// TIA Portal V18 export
FUNCTION_BLOCK "FS_Room1"   // FB2, F_LAD
{ S7_Optimized_Access := 'TRUE' }
VERSION : 0.1
// 急停：2NC 硬件组态配置
// 1,急停故障
// 2,急停已恢复，需要确认
// 
// 
// 钥匙：1NC+1NO
// 1，钥匙电磁基座信号不匹配
// 2，基座信号正常，需要确认
// 3，安全钥匙2个电磁基座信号一致性故障，均显示插入
// 4，安全钥匙2个电磁基座信号一致性正常，需要确认
// 
// 门：2NC时关闭
// 1，门信号不一致，需要同时开同时关闭
// stored: AutoNumber true, IsIECCheckEnabled false, UDAEnableTagReadback false
   VAR_INPUT
      ACK : Bool;
   END_VAR
   VAR_OUTPUT
      ES_OK : Bool;
   END_VAR
   VAR
      EStop1 { S7_SetPoint := 'True'} : ESTOP1;
      EStop2 { S7_SetPoint := 'True'} : ESTOP1;
      EStop3 { S7_SetPoint := 'True'} : ESTOP1;
      EStop4 { S7_SetPoint := 'True'} : ESTOP1;
      EStop5 { S7_SetPoint := 'True'} : ESTOP1;
      EStop6 : ESTOP1;
      door : SFDOOR;
      Key : SFDOOR;
      KeyControl : SFDOOR;
      Door_Timer : TON;
      Key1 : TON;
      KeyControl1 : TON;
      Key_InDoor : Bool;
      Key_InControl : Bool;
   END_VAR
BEGIN

REGION Network 1: E-Stop1
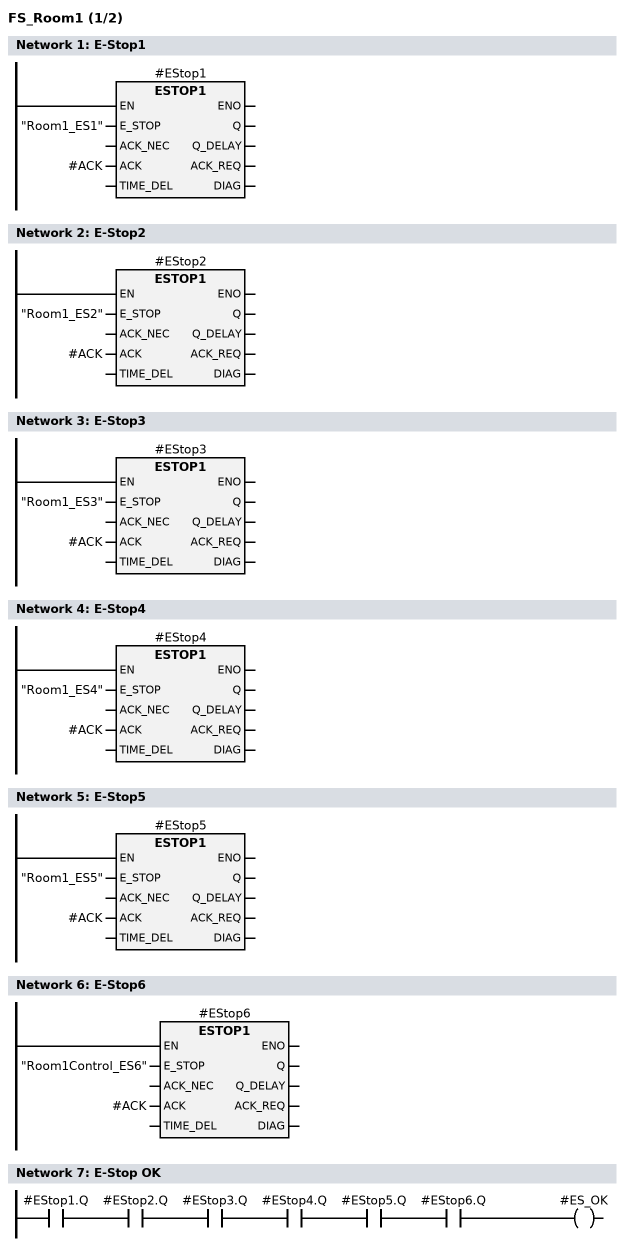
   RUNG wire#powerrail
      #EStop1.ESTOP1(E_STOP := "Room1_ES1", ACK_NEC :=, ACK := #ACK, TIME_DEL :=, Q =>, Q_DELAY =>, ACK_REQ =>, DIAG =>)
   END_RUNG
   // the same network as SCL:
   #EStop1(E_STOP := "Room1_ES1", ACK := #ACK);   // ESTOP1
END_REGION

REGION Network 2: E-Stop2
   RUNG wire#powerrail
      #EStop2.ESTOP1(E_STOP := "Room1_ES2", ACK_NEC :=, ACK := #ACK, TIME_DEL :=, Q =>, Q_DELAY =>, ACK_REQ =>, DIAG =>)
   END_RUNG
   // the same network as SCL:
   #EStop2(E_STOP := "Room1_ES2", ACK := #ACK);   // ESTOP1
END_REGION

REGION Network 3: E-Stop3
   RUNG wire#powerrail
      #EStop3.ESTOP1(E_STOP := "Room1_ES3", ACK_NEC :=, ACK := #ACK, TIME_DEL :=, Q =>, Q_DELAY =>, ACK_REQ =>, DIAG =>)
   END_RUNG
   // the same network as SCL:
   #EStop3(E_STOP := "Room1_ES3", ACK := #ACK);   // ESTOP1
END_REGION

REGION Network 4: E-Stop4
   RUNG wire#powerrail
      #EStop4.ESTOP1(E_STOP := "Room1_ES4", ACK_NEC :=, ACK := #ACK, TIME_DEL :=, Q =>, Q_DELAY =>, ACK_REQ =>, DIAG =>)
   END_RUNG
   // the same network as SCL:
   #EStop4(E_STOP := "Room1_ES4", ACK := #ACK);   // ESTOP1
END_REGION

REGION Network 5: E-Stop5
   RUNG wire#powerrail
      #EStop5.ESTOP1(E_STOP := "Room1_ES5", ACK_NEC :=, ACK := #ACK, TIME_DEL :=, Q =>, Q_DELAY =>, ACK_REQ =>, DIAG =>)
   END_RUNG
   // the same network as SCL:
   #EStop5(E_STOP := "Room1_ES5", ACK := #ACK);   // ESTOP1
END_REGION

REGION Network 6: E-Stop6
   RUNG wire#powerrail
      #EStop6.ESTOP1(E_STOP := "Room1Control_ES6", ACK_NEC :=, ACK := #ACK, TIME_DEL :=, Q =>, Q_DELAY =>, ACK_REQ =>, DIAG =>)
   END_RUNG
   // the same network as SCL:
   #EStop6(E_STOP := "Room1Control_ES6", ACK := #ACK);   // ESTOP1
END_REGION

REGION Network 7: E-Stop OK
   RUNG wire#powerrail
      Contact( #EStop1.Q )
      Contact( #EStop2.Q )
      Contact( #EStop3.Q )
      Contact( #EStop4.Q )
      Contact( #EStop5.Q )
      Contact( #EStop6.Q )
      Coil( #ES_OK )
   END_RUNG
   // the same network as SCL:
   #ES_OK := #EStop1.Q AND #EStop2.Q AND #EStop3.Q AND #EStop4.Q AND #EStop5.Q AND #EStop6.Q;
END_REGION

REGION Network 8: door
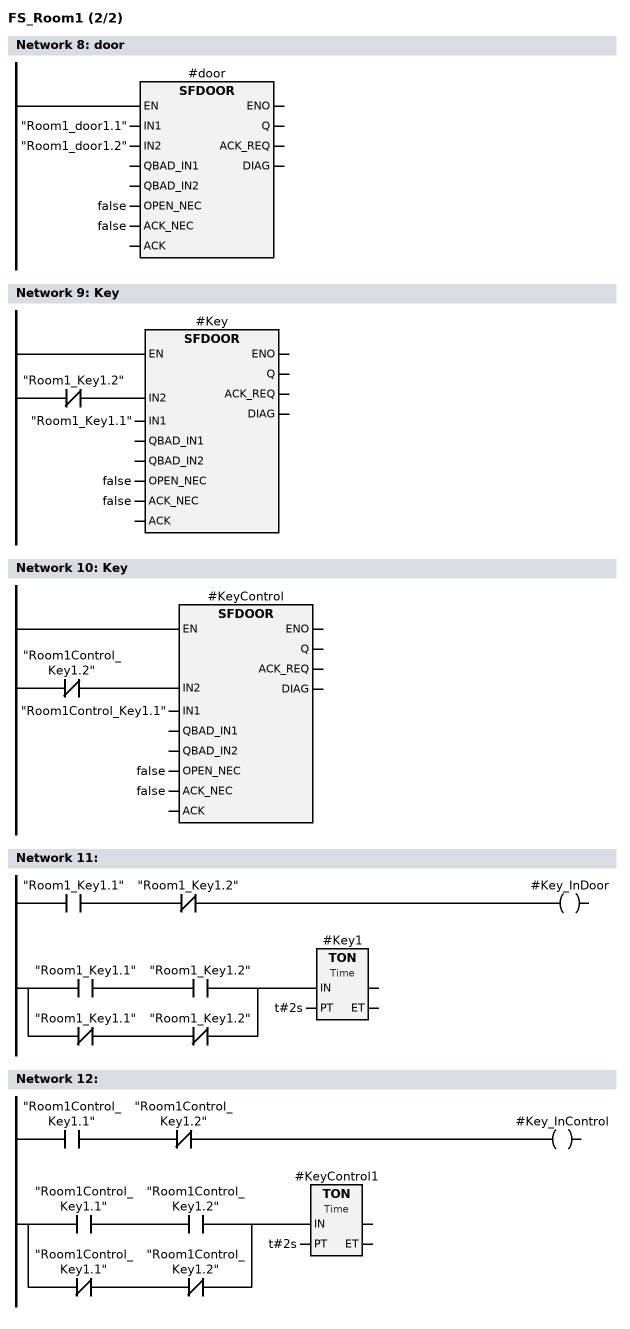
   RUNG wire#powerrail
      #door.SFDOOR(IN1 := "Room1_door1.1", IN2 := "Room1_door1.2", QBAD_IN1 :=, QBAD_IN2 :=, OPEN_NEC := false, ACK_NEC := false, ACK :=, Q =>, ACK_REQ =>, DIAG =>)
   END_RUNG
   // the same network as SCL:
   #door(IN1 := "Room1_door1.1", IN2 := "Room1_door1.2", OPEN_NEC := false, ACK_NEC := false);   // SFDOOR
END_REGION

REGION Network 9: Key
   RUNG wire#powerrail
      #Key.SFDOOR(IN2 := wire#w1, IN1 := "Room1_Key1.1", QBAD_IN1 :=, QBAD_IN2 :=, OPEN_NEC := false, ACK_NEC := false, ACK :=, Q =>, ACK_REQ =>, DIAG =>)
   END_RUNG
   RUNG wire#powerrail
      I_Contact( "Room1_Key1.2" )
   END_RUNG wire#w1
   // the same network as SCL:
   #Key(IN2 := NOT "Room1_Key1.2", IN1 := "Room1_Key1.1", OPEN_NEC := false, ACK_NEC := false);   // SFDOOR
END_REGION

REGION Network 10: Key
   RUNG wire#powerrail
      #KeyControl.SFDOOR(IN2 := wire#w1, IN1 := "Room1Control_Key1.1", QBAD_IN1 :=, QBAD_IN2 :=, OPEN_NEC := false, ACK_NEC := false, ACK :=, Q =>, ACK_REQ =>, DIAG =>)
   END_RUNG
   RUNG wire#powerrail
      I_Contact( "Room1Control_Key1.2" )
   END_RUNG wire#w1
   // the same network as SCL:
   #KeyControl(IN2 := NOT "Room1Control_Key1.2",   // SFDOOR
               IN1 := "Room1Control_Key1.1",
               OPEN_NEC := false,
               ACK_NEC := false);
END_REGION

REGION Network 11
   RUNG wire#powerrail
      Contact( "Room1_Key1.1" )
      I_Contact( "Room1_Key1.2" )
      Coil( #Key_InDoor )
   END_RUNG
   RUNG wire#powerrail
      Contact( "Room1_Key1.1" )
      Contact( "Room1_Key1.2" )
      wire#w1
      { S7_Templates := "[time_type := Time, codedbool_type := DInt]" } #Key1.TON(pt := t#2s, et =>)
   END_RUNG
   RUNG wire#powerrail
      I_Contact( "Room1_Key1.1" )
      I_Contact( "Room1_Key1.2" )
   END_RUNG wire#w1
   // the same network as SCL:
   #Key_InDoor := "Room1_Key1.1" AND NOT "Room1_Key1.2";
   #Key1.TON(IN := ("Room1_Key1.1" AND "Room1_Key1.2") OR (NOT "Room1_Key1.1" AND NOT "Room1_Key1.2"),
             PT := t#2s);
END_REGION

REGION Network 12
   RUNG wire#powerrail
      Contact( "Room1Control_Key1.1" )
      I_Contact( "Room1Control_Key1.2" )
      Coil( #Key_InControl )
   END_RUNG
   RUNG wire#powerrail
      Contact( "Room1Control_Key1.1" )
      Contact( "Room1Control_Key1.2" )
      wire#w1
      { S7_Templates := "[time_type := Time, codedbool_type := DInt]" } #KeyControl1.TON(pt := t#2s, et =>)
   END_RUNG
   RUNG wire#powerrail
      I_Contact( "Room1Control_Key1.1" )
      I_Contact( "Room1Control_Key1.2" )
   END_RUNG wire#w1
   // the same network as SCL:
   #Key_InControl := "Room1Control_Key1.1" AND NOT "Room1Control_Key1.2";
   #KeyControl1.TON(IN := ("Room1Control_Key1.1" AND "Room1Control_Key1.2") OR (NOT "Room1Control_Key1.1" AND NOT "Room1Control_Key1.2"),
                    PT := t#2s);
END_REGION
END_FUNCTION_BLOCK
